Omron Sysmac Studio project Teste_Modbus (Sysmac Studio 1.64.0.64008, StandardProject)

# Controller new_Controller_0: NX102-1020 version 1.33
Units and slaves: Unit 1 : NX-PF0730 (N1); Unit 2 : NX-ID5442 (N2); Unit 3 : NX-OD5256 (N3); Unit 5 : NX-SID800 (N5); Unit 6 : NX-SOD400 (N6)
Task PrimaryTask (priority 4, period or condition 2000): Program0

VAR_GLOBAL
    Server : _sSOCKET;
    aDataSnd : ARRAY[0..9] OF WORD;
    aDataRcv : ARRAY[0..9] OF WORD;
END_VAR

(* Program Program0: safety or other program stored in binary form, left out *)

PROGRAM Program0
VAR
    bConnect : BOOL;
    ModBusTeste : ModbusTCPCmd;
    ModBusComm : SktTCPConnect;
    Buffer : SktClearBuf;
    bCmd : BOOL;
    CloseComm : SktClose;
    bClose : BOOL;
    tmrConnect : TON;
    bWrite : BOOL;
    ModWrite : ModbusTCPWrite;
    SetWriteCMD : _sMODBUS_WRITE;
    bRead : BOOL;
    ModRead : ModbusTCPRead;
    SetReadCmd : _sMODBUS_READ;
END_VAR
VAR_EXTERNAL
    Server : _sSOCKET;
    aDataRcv : ARRAY[0..9] OF WORD;
END_VAR
VAR_EXTERNAL CONSTANT
    _EIP1_EtnOnlineSta : BOOL;
END_VAR
VAR_EXTERNAL
    aDataSnd : ARRAY[0..9] OF WORD;
END_VAR
VAR
    _e1 : R_TRIG;
    _p2 : BOOL;
END_VAR

(* Section ModBus_Master: ladder, written here as Structured Text *)

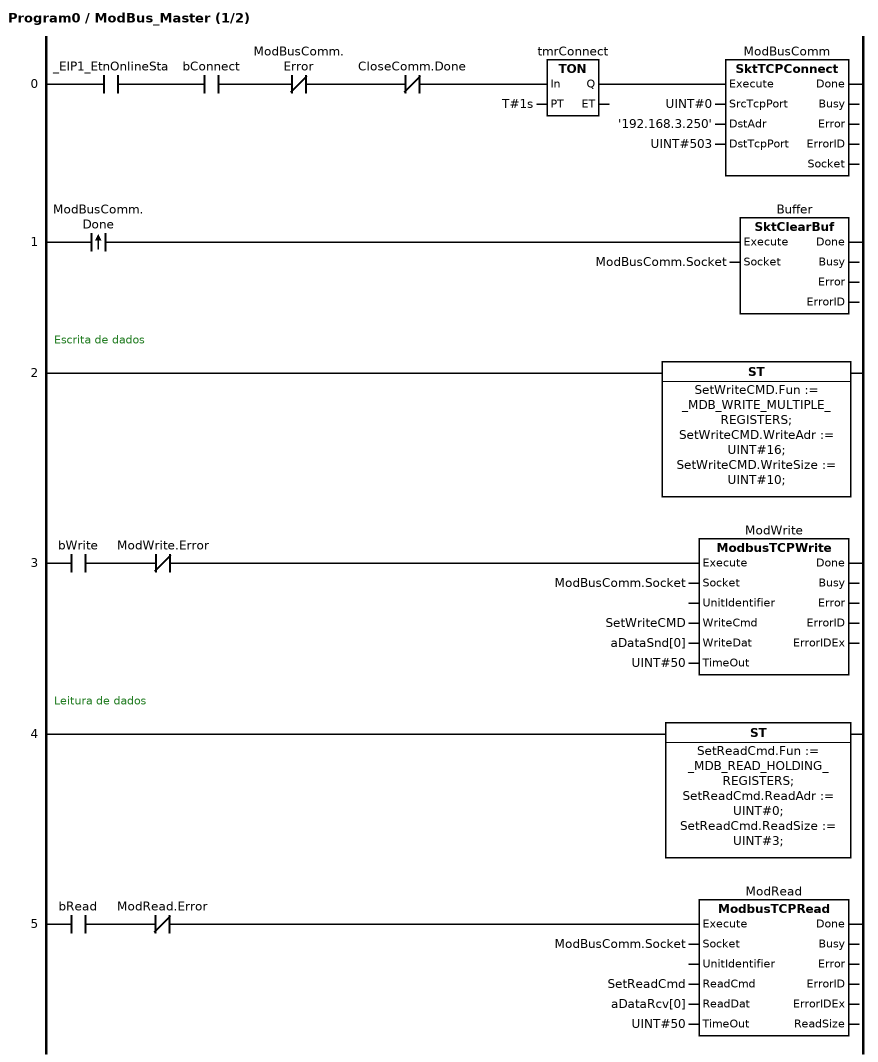
(* Rung 0 *)
tmrConnect(In := _EIP1_EtnOnlineSta AND bConnect AND NOT ModBusComm.Error AND NOT CloseComm.Done, PT := T#1s);
ModBusComm(Execute := tmrConnect.Q, SrcTcpPort := UINT#0, DstAdr := '192.168.3.250', DstTcpPort := UINT#503);
(* Rung 1 *)
_e1(CLK := ModBusComm.Done);
Buffer(Execute := _e1.Q, Socket := ModBusComm.Socket);
(* Rung 2: Escrita de dados *)
SetWriteCMD.Fun := _MDB_WRITE_MULTIPLE_REGISTERS;
SetWriteCMD.WriteAdr := UINT#16;
SetWriteCMD.WriteSize := UINT#10;
(* Rung 3 *)
ModWrite(Execute := bWrite AND NOT ModWrite.Error, Socket := ModBusComm.Socket, WriteCmd := SetWriteCMD, WriteDat := aDataSnd[0], TimeOut := UINT#50);
(* Rung 4: Leitura de dados *)
SetReadCmd.Fun := _MDB_READ_HOLDING_REGISTERS;
SetReadCmd.ReadAdr := UINT#0;
SetReadCmd.ReadSize := UINT#3;
(* Rung 5 *)
ModRead(Execute := bRead AND NOT ModRead.Error, Socket := ModBusComm.Socket, ReadCmd := SetReadCmd, ReadDat := aDataRcv[0], TimeOut := UINT#50);

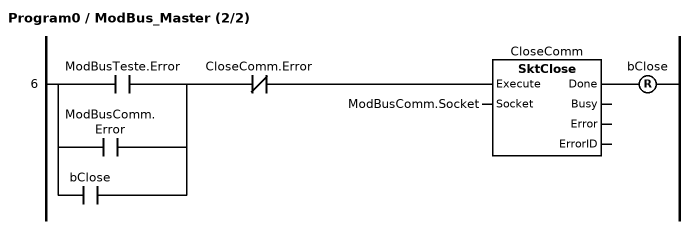
(* Rung 6 *)
_p2 := (ModBusTeste.Error OR ModBusComm.Error OR bClose) AND NOT CloseComm.Error;
CloseComm(Execute := _p2, Socket := ModBusComm.Socket);
IF CloseComm.Done THEN bClose := FALSE; END_IF;
END_PROGRAM